TYPE g_E:
    (LIT1_g_E, LIT2_g_E);
END_TYPE

(* stored: ProductVersion 3.1.0.18, Version 1.1.0.1 *)
